KUKA KRL data list: vw_vm_currlim.dat

&ACCESS RV
&REL 10
&COMMENT KS_17.3_VW
&PARAM DISKPATH = VW_User
&PARAM TPVW_VERSION = 8.1.8
&PARAM EDITMASK = vw_usr_r
DEFDAT  vw_vm_currlim PUBLIC
; KUKA library for vectormove current Limitation
;
; configured force limitation [N]
GLOBAL INT nForceLimitationVM_Prog=50
GLOBAL INT nForceLimitationVM_Teach=50
;
GLOBAL INT starttime=1715142655
;
; configured duration active phase [ms]
GLOBAL INT nActiveTimeVectormove=350
; configured length of active phase [1/10ms]
GLOBAL INT nActivePathVectormove=25
;
FRAME A1Pos={X 1956.27002,Y 1682.67004,Z 4114.7998,A 89.8820038,B 110.920998,C 0.305999994}
FRAME A2Pos={X 1615.9917,Y 2294.84717,Z 3818.86914,A -176.964462,B 9.02532005,C 111.195511}
FRAME A3Pos={X 1957.56104,Y 3533.5708,Z 3404.87158,A 74.5841827,B 17.8583584,C 75.3347626}
FRAME A4Pos={X 862.867065,Y 3042.05884,Z 3397.06055,A -155.82016,B 0.372953266,C 112.952522}
FRAME A5Pos={X 862.867065,Y 3042.05884,Z 3397.06055,A -155.82016,B 0.372953266,C -172.739944}
FRAME A6Pos={X 879.495361,Y 3004.94214,Z 3402.2417,A -137.416809,B 68.0746002,C -160.218597}
FRAME A1PosInv={X 0.0,Y 0.0,Z 0.0,A 0.0,B 0.0,C 0.0}
FRAME A2PosInv={X -350.000,Y 0.0,Z -675.000,A 3.31803567E-05,B 0.0,C 0.0}
FRAME A3PosInv={X -1640.50269,Y 2.46989366E-05,Z 580.975220,A 179.999908,B 67.5811386,C 179.999924}
FRAME A4PosInv={X -1114.60974,Y 1.62659217E-05,Z -1738.24341,A 3.05176363E-05,B 0.105171204,C 5.60164892E-08}
FRAME A5PosInv={X -1114.60974,Y 96.2042465,Z -1735.57910,A 0.00585124735,B 0.105008326,C 3.17269945}
FRAME A6PosInv={X 2061.49023,Y 137.204269,Z -69.6282959,A 179.988510,B -59.3304100,C -176.817444}
FRAME ArmVector={X 1125.24707,Y -1093.29468,Z -3463.95801,A 0.0,B 0.0,C 0.0}
FRAME AxisVector={X 0.00732421875,Y 0.934082031,Z -0.356933594,A 0.0,B 0.0,C 0.0}
FRAME AxisPerpVector={X 670.0,Y -318.670898,Z -35.0,A 0.0,B 0.0,C 0.0}

FRAME FramePosAct={X 3081.51709,Y 589.375427,Z 650.841919,A 108.974503,B 12.5054197,C -82.5577011}
E6AXIS AxisAxisAct={A1 -80.4487686,A2 -104.442787,A3 127.20343,A4 74.3075409,A5 68.8793259,A6 98.2319794,E1 9.08152485,E2 0.0,E3 0.0,E4 0.0,E5 0.0,E6 0.0}
E6AXIS AxisForceDirection={A1 -80.3487701,A2 -104.442787,A3 127.20343,A4 74.3075409,A5 68.8793259,A6 98.2319794,E1 9.08152485,E2 0.0,E3 0.0,E4 0.0,E5 0.0,E6 0.0}
FRAME FrameTCPDirection={X -0.946777344,Y -0.295898438,Z 0.126464844,A 0.0,B 0.0,C 0.0}
FRAME FrameForceDirection={X 0.852539063,Y -2.09936523,Z -2.21899414,A 0.0,B 0.0,C 0.0}

INT lnLeadingAxis=1
REAL rDistAxisToTCP=3.80269384
REAL rDistAxisToTCPPerp=3.79612494
REAL rDistAxisinAxisDir=0.223421827
REAL rAngleArmAxis=86.6317291
REAL rAngleArmTCP=64.5931854
REAL lrAverageTorque=-2333.66504
REAL rForceAtTCP=-41.206749
REAL rAngleForceTCP=81.5395355
REAL rForceTCPDirection=-6.06262255
REAL lrForceLimit=50.0
REAL rAdditionalTorque=1290.08496
REAL lrTorqueFactor=-8.24725628

REAL rVector1[3]
rVector1[1]=0.268816859
rVector1[2]=-0.661957681
rVector1[3]=-0.699678242
REAL rVector2[3]
rVector2[1]=-0.946807384
rVector2[2]=-0.295907825
rVector2[3]=0.126468852

ENDDAT
